FUNCTION_BLOCK FieldsToServiceRegistryEntry (* Translate individual fields to a Service Registry type *)
  (* Standard: 61499-2; Description: Copyright (c) 2018 fortiss GmbH This program and the accompanying materials are made available under the terms of the Eclipse Public License 2.0 which is available at https://www.eclipse.org/legal/epl-2.0/ SPDX-License-Identifier: EPL-2.0 *)
  (* Version 1.0, 2018-09-21, Jose Cabral, fortiss GmbH *)
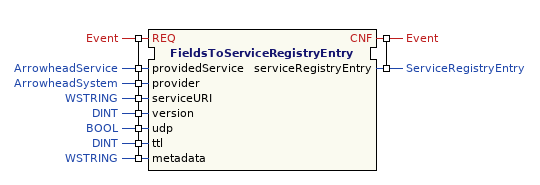
  EVENT_INPUT
    REQ WITH metadata, ttl, udp, version, serviceURI, provider, providedService; (* Create service registry entry *)
  END_EVENT
  EVENT_OUTPUT
    CNF WITH serviceRegistryEntry; (* Service registry entry created *)
  END_EVENT
  VAR_INPUT
    providedService : ArrowheadService; (* The Arrowhead Service object that is provided (SD and supported IDD-s) *)
    provider : ArrowheadSystem; (* ArrowheadSystem that is providing the Service *)
    serviceURI : WSTRING; (* The URL subpath of the Service within the address:port of the Provider *)
    version : DINT; (* The version numbering of the Service provided *)
    udp : BOOL; (* True, if the service is provided via UDP. By default, it is false *)
    ttl : DINT; (* Service validity time period expressed in seconds. This gets converted to a date-time, and stored in the database *)
    metadata : WSTRING; (* Metadata belonging to a service/provider pair *)
  END_VAR
  VAR_OUTPUT
    serviceRegistryEntry : ServiceRegistryEntry; (* Created Service Registry entry *)
  END_VAR
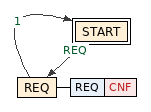
  EC_STATES
    START; (* Initial State *)
    REQ : REQ -> CNF; (* Normal execution *)
  END_STATES
  EC_TRANSITIONS
    START TO REQ := REQ;
    REQ TO START := 1;
  END_TRANSITIONS
  ALGORITHM REQ IN ST: (* Normally executed algorithm *)
serviceRegistryEntry.providedService := providedService;
serviceRegistryEntry.provider := provider;
serviceRegistryEntry.serviceURI := serviceURI;
serviceRegistryEntry.version := version;
serviceRegistryEntry.udp := udp;
serviceRegistryEntry.ttl := ttl;
serviceRegistryEntry.metadata := metadata;
  END_ALGORITHM
END_FUNCTION_BLOCK
